// Mitsubishi GX Works2 project: plcV3   PLC: FX3G

TYPE ST_INTENS : STRUCT
  RECIRC : INT;
  ASPER : INT;
END_STRUCT END_TYPE

// global labels: GVL
VAR_GLOBAL
  g_iIntensity AT D500 : INT;  (* Интенсивность: 0=Слабо, 1=Нормально, 2=Интенсивно (настройка HMI) *)
  g_iToutAsper AT D501 : INT;  (* Мин. t улицы для аспирации, °C×10 (по умолч. 30 = 3.0°C) *)
  g_iToutHeat AT D502 : INT;  (* Мин. t улицы для подогрева, °C×10 (по умолч. 50 = 5.0°C) *)
  g_iPreheatTime AT D504 : INT;  (* Время предподогрева заслонок, мин (по умолч. 3) *)
  g_iManualAspMin AT D506 : INT;  (* Время ручной аспирации, мин (ввод оператора, по умолч. 5) *)
  g_iPreheatLeft AT D507 : INT;  (* Текущее время подогрева, мин (обратный отсчёт для HMI) *)
  g_iAutoResetDelay AT D508 : INT;  (* Задержка автосброса, мин (по умолч. 60) *)
  g_iTprodMax AT D509 : INT;  (* Макс. температура продукта, °C×10 (задаётся оператором) *)
  g_iHmin AT D510 : INT;  (* Мин. влажность, %×10 (задаётся оператором) *)
  g_iCorrTout AT D511 : INT;  (* Коррекция t улицы (Pt100), °C×10 (настройка HMI) *)
  g_iCorrTprod1 AT D512 : INT;  (* Коррекция щупа 1 (Pt100), °C×10 (настройка HMI) *)
  g_iCorrTprod2 AT D513 : INT;  (* Коррекция щупа 2 (Pt100), °C×10 (настройка HMI) *)
  g_iCorrTprod3 AT D514 : INT;  (* Коррекция щупа 3 (Pt100), °C×10 (настройка HMI) *)
  g_iCorrTprod4 AT D515 : INT;  (* Коррекция щупа 4 (Pt100), °C×10 (настройка HMI) *)
  g_iMbAddr AT D516 : INT;  (* Modbus slave: адрес ПЛК (1..247, по умолч. 1) *)
  g_iValveTime AT D517 : INT;  (* Время хода клапана, с (по умолч. 120) *)
  g_iProgress AT D518 : INT;  (* Время исполнения в % 0-100 *)
  g_iLeftTime AT D519 : INT;  (* Сколько минут осталось обратный отсчет *)
  g_iFun1State AT D520 : INT;  (* Состояние вентилятора 1 *)
  g_iFun2State AT D521 : INT;  (* Состояние вентилятора 2 *)
  g_iFun3State AT D522 : INT;  (* Состояние вентилятора 3 *)
  g_iFun4State AT D523 : INT;  (* Состояние вентилятора 4 *)
  g_iFun5State AT D524 : INT;  (* Состояние вентилятора 5 *)
  g_iFun6State AT D525 : INT;  (* Состояние вентилятора 6 *)
  g_iFun7State AT D526 : INT;  (* Состояние вентилятора 7 *)
  g_iFun8State AT D527 : INT;  (* Состояние вентилятора 8 *)
  g_iFun9State AT D528 : INT;  (* Состояние вентилятора 9 *)
  g_iFun10State AT D529 : INT;  (* Состояние вентилятора 10 *)
  g_iModeDisp AT D530 : INT;  (* Детальный режим для HMI: 0=Выкл, 1=Авто, 2=Продувка, 3=Аспирацияб, 4=Прогрев клапанов, 5-ручная аспирация *)
  g_iRecircLeft AT D531 : INT;  (* Отсчёт рециркуляции, мин *)
  g_iAspLeft AT D532 : INT;  (* Обратный отсчёт аспирации *)
  g_iAlarmCount AT D533 : INT;  (* Количество активных тревог *)
  g_iStep AT D534 : INT;  (* Состояние автомата (0/2/50/100/200/210/300, отладка) *)
  g_iModeCoarse AT D535 : INT;  (* Грубый режим по переключателю: 0=Выкл, 1=Авто, 2=Продувка *)
  g_iCurWait AT D536 : INT;  (* Текущее время ожидания в авто режиме в выбраной интенсивности *)
  g_iCurAsper AT D537 : INT;  (* Текущее время аспирации в авто режиме в выбраной интенсивности *)
  g_iAlarmPack1 AT D550 : INT;  (* Упакованные тревоги 0-15 (AM_PACK) *)
  g_iAlarmPack2 AT D551 : INT;  (* Упакованные тревоги 16-27 (AM_PACK) *)
  g_iAlarmPack3 AT D552 : INT;  (* Упакованные тревоги 32-33 (AM_PACK) *)
  g_xCmdFanH1 AT M500 : BOOL;  (* Команда напорный вентилятор 1 *)
  g_xCmdFanH2 AT M501 : BOOL;  (* Команда напорный вентилятор 2 *)
  g_xCmdFanH3 AT M502 : BOOL;  (* Команда напорный вентилятор 3 *)
  g_xCmdFanH4 AT M503 : BOOL;  (* Команда напорный вентилятор 4 *)
  g_xCmdFanH5 AT M504 : BOOL;  (* Команда напорный вентилятор 5 *)
  g_xCmdFanH6 AT M505 : BOOL;  (* Команда напорный вентилятор 6 *)
  g_xCmdFanR1 AT M506 : BOOL;  (* Команда разгонный вентилятор 1 *)
  g_xCmdFanR2 AT M507 : BOOL;  (* Команда разгонный вентилятор 2 *)
  g_xCmdFanR3 AT M508 : BOOL;  (* Команда разгонный вентилятор 3 *)
  g_xCmdFanR4 AT M509 : BOOL;  (* Команда разгонный вентилятор 4 *)
  g_xCmdValveIn1 AT M510 : BOOL;  (* Команда открыть клапан приток 1 *)
  g_xCmdValveIn2 AT M511 : BOOL;  (* Команда открыть клапан приток 2 *)
  g_xCmdValveOut1 AT M512 : BOOL;  (* Команда открыть клапан сброс 1 *)
  g_xCmdValveOut2 AT M513 : BOOL;  (* Команда открыть клапан сброс 2 *)
  g_xCmdValveRec1 AT M514 : BOOL;  (* Команда открыть клапан рециркуляция 1 *)
  g_xCmdValveRec2 AT M515 : BOOL;  (* Команда открыть клапан рециркуляция 2 *)
  g_xCmdHeat AT M516 : BOOL;  (* Подогрев клапана приток *)
  g_xCoolerWorks AT M517 : BOOL;  (* Холод работает *)
  g_xIsAuto AT M518 : BOOL;  (* Автоматический режим *)
  g_xAspirNow AT M519 : BOOL;  (* Сейчас идет асперация *)
  g_xCmdCoolerStop AT M520 : BOOL;  (* Команда «Остановить холод» (Y00) *)
  g_xManualAspActive AT M521 : BOOL;  (* Ручная аспирация выполняется *)
  g_xManualAspCmd AT M522 : BOOL;  (* Кнопка HMI: ручная аспирация (фронт) *)
  g_xAlarmResetHmi AT M523 : BOOL;  (* Кнопка HMI: сброс тревог (фронт) *)
  g_xModeManual AT M524 : BOOL;  (* Ручной режим если ни какой режим не выбран на входах *)
  g_xAutoReset AT M525 : BOOL;  (* Автосброс тревог: TRUE=вкл, FALSE=выкл (по умолч. выкл) *)
  g_xMbApply AT M526 : BOOL;  (* Кнопка HMI: применить настройки Modbus (фронт) *)
  g_xValveIn AT M527 : BOOL;  (* Кнопка HMI: применить настройки Modbus (фронт) *)
  g_xValveOut AT M528 : BOOL;  (* Кнопка HMI: применить настройки Modbus (фронт) *)
  g_xValveRecycle AT M529 : BOOL;  (* Кнопка HMI: применить настройки Modbus (фронт) *)
  g_xRecycleFlow AT M530 : BOOL;  (* Поток идет рециркуляция *)
  g_xAnyAlarm AT M550 : BOOL;  (* Есть активная тревога (AM_HAS_ALARMS) *)
  g_xAnyBlock AT M551 : BOOL;  (* Есть блокирующая тревога (AM_IS_BLOCK) *)
END_VAR
VAR_GLOBAL CONSTANT
  c_AM_ALARMS_NUM : INT := 33;  (* Верхняя граница массива AM_ALARMS (34 тревоги, ID 0..33) *)
  c_AM_EVENTS_NUM : INT;  (* Верхняя граница массива AM_EVENTS (события не используются) *)
END_VAR
VAR_GLOBAL
  astIntens : ARRAY [0..2] OF ST_INTENS;  (* Уровени интенсивности. Назначить D540 как главный *)
  AM_ALARMS : ARRAY [0..33] OF ST_AM_ALARM;  (* Хранилище тревог AlarmManager (объявляет приложение, V206+) *)
  AM_EVENTS : ARRAY [0..0] OF ST_AM_EVENT;  (* Хранилище событий AlarmManager (объявляет приложение, V206+) *)
  g_iTCorrection AT D538 : INT;  (* Корекция температуры *)
END_VAR

// global labels: IO
VAR_GLOBAL
  DI_ModeAuto AT X000 : BOOL;  (* Переключатель режима — «Авто» / ШУК-D1 *)
  DI_ModePurge AT X001 : BOOL;  (* Переключатель режима — «Продувка» / ШУК-D1 *)
  DI_PhaseFault AT X002 : BOOL;  (* Реле контроля фаз — ошибка фазировки / ШУК-D1 *)
  DI_CoolerRun AT X003 : BOOL;  (* Охладитель в работе (идёт охлаждение) / ШУК-D1 *)
  DI_VlvIn1Close AT X004 : BOOL;  (* Концевик клапана приток №1 — закрыт (НО) / ШУК-D1 *)
  DI_VlvIn2Close AT X005 : BOOL;  (* Концевик клапана приток №2 — закрыт (НО) / ШУК-D1 *)
  DI_FanHFb1 AT X006 : BOOL;  (* Обратная связь напорного вентилятора №1 (пускатель/тепловое реле) / ШУК-D1 *)
  DI_FanHFb2 AT X007 : BOOL;  (* Обратная связь напорного вентилятора №2 (пускатель/тепловое реле) / ШУК-D1 *)
  DI_FanHFb3 AT X010 : BOOL;  (* Обратная связь напорного вентилятора №3 (пускатель/тепловое реле) / ШУК-D1 *)
  DI_FanHFb4 AT X011 : BOOL;  (* Обратная связь напорного вентилятора №4 (пускатель/тепловое реле) / ШУК-D1 *)
  DI_FanHFb5 AT X012 : BOOL;  (* Обратная связь напорного вентилятора №5 (пускатель/тепловое реле) / ШУК-D1 *)
  DI_FanHFb6 AT X013 : BOOL;  (* Обратная связь напорного вентилятора №6 (пускатель/тепловое реле) / ШУК-D1 *)
  DI_VlvOut1Close AT X020 : BOOL;  (* Концевик клапана сброс №1 — закрыт (НО) / ШУК-D2 *)
  DI_VlvOut2Close AT X021 : BOOL;  (* Концевик клапана сброс №2 — закрыт (НО) / ШУК-D2 *)
  DI_VlvRec1Close AT X022 : BOOL;  (* Концевик клапана рециркуляция №1 — закрыт (НО) / ШУК-D2 *)
  DI_VlvRec2Close AT X023 : BOOL;  (* Концевик клапана рециркуляция №2 — закрыт (НО) / ШУК-D2 *)
  DI_VlvIn1Open AT X024 : BOOL;  (* Концевик клапана приток №1 — открыт / ШУК-D2 *)
  DI_VlvIn2Open AT X025 : BOOL;  (* Концевик клапана приток №2 — открыт / ШУК-D2 *)
  DI_VlvOut1Open AT X026 : BOOL;  (* Концевик клапана сброс №1 — открыт / ШУК-D2 *)
  DI_VlvOut2Open AT X027 : BOOL;  (* Концевик клапана сброс №2 — открыт / ШУК-D2 *)
  DI_VlvRec1Open AT X030 : BOOL;  (* Концевик клапана рециркуляция №1 — открыт / ШУК-D2 *)
  DI_VlvRec2Open AT X031 : BOOL;  (* Концевик клапана рециркуляция №2 — открыт / ШУК-D2 *)
  DI_Flow1 AT X032 : BOOL;  (* Реле давления №1 — поток есть / ШУК-D2; РД-ДД200, контакт НЗ *)
  DI_Flow2 AT X033 : BOOL;  (* Реле давления №2 — поток есть / ШУК-D2; РД-ДД200, контакт НЗ *)
  DI_Flow3 AT X034 : BOOL;  (* Реле давления №3 — поток есть / ШУК-D2; РД-ДД200, контакт НЗ *)
  DI_Flow4 AT X035 : BOOL;  (* Реле давления №4 — поток есть / ШУК-D2; РД-ДД200, контакт НЗ *)
  DI_Flow5 AT X036 : BOOL;  (* Реле давления №5 — поток есть / ШУК-D2; РД-ДД200, контакт НЗ *)
  DI_Flow6 AT X037 : BOOL;  (* Реле давления №6 — поток есть / ШУК-D2; РД-ДД200, контакт НЗ *)
  DO_CoolerStop AT Y000 : BOOL;  (* Остановить холод (1 = запрет охлаждения, 0 = разрешение) / ШУК-D1 *)
  DO_FanR1 AT Y002 : BOOL;  (* Разгонный вентилятор №1 (220 В, без обратной связи) / ШУК-D1 *)
  DO_FanR2 AT Y003 : BOOL;  (* Разгонный вентилятор №2 (220 В, без обратной связи) / ШУК-D1 *)
  DO_FanR3 AT Y004 : BOOL;  (* Разгонный вентилятор №3 (220 В, без обратной связи) / ШУК-D1 *)
  DO_FanR4 AT Y005 : BOOL;  (* Разгонный вентилятор №4 (220 В, без обратной связи) / ШУК-D1 *)
  DO_FanH1 AT Y006 : BOOL;  (* Напорный вентилятор №1 (2.2 кВт, 380 В) / ШУК-D1 *)
  DO_FanH2 AT Y007 : BOOL;  (* Напорный вентилятор №2 (2.2 кВт, 380 В) / ШУК-D1 *)
  DO_FanH3 AT Y010 : BOOL;  (* Напорный вентилятор №3 (2.2 кВт, 380 В) / ШУК-D1 *)
  DO_FanH4 AT Y011 : BOOL;  (* Напорный вентилятор №4 (2.2 кВт, 380 В) / ШУК-D1 *)
  DO_FanH5 AT Y012 : BOOL;  (* Напорный вентилятор №5 (2.2 кВт, 380 В) / ШУК-D1 *)
  DO_FanH6 AT Y013 : BOOL;  (* Напорный вентилятор №6 (2.2 кВт, 380 В) / ШУК-D1 *)
  DO_HeatVlv AT Y020 : BOOL;  (* Подогрев клапана (ТЭН 4x300 Вт) / ШУК-D3 *)
  DO_VlvIn1Open AT Y024 : BOOL;  (* Открыть клапан приток №1 (Belimo LF230, пружина закрывает) / ШУК-D3 *)
  DO_VlvIn2Open AT Y025 : BOOL;  (* Открыть клапан приток №2 (Belimo LF230, пружина закрывает) / ШУК-D3 *)
  DO_VlvOut1Open AT Y026 : BOOL;  (* Открыть клапан сброс №1 (Belimo LF230, пружина закрывает) / ШУК-D3 *)
  DO_VlvOut2Open AT Y027 : BOOL;  (* Открыть клапан сброс №2 (Belimo LF230, пружина закрывает) / ШУК-D3 *)
  DO_VlvRec1Open AT Y030 : BOOL;  (* Открыть клапан рециркуляция №1 (Belimo LF230, пружина закрывает) / ШУК-D3 *)
  DO_VlvRec2Open AT Y031 : BOOL;  (* Открыть клапан рециркуляция №2 (Belimo LF230, пружина закрывает) / ШУК-D3 *)
  DO_LampGreen AT Y032 : BOOL;  (* Световая колонна — зелёный / ШУК-D3 *)
  DO_LampRed AT Y033 : BOOL;  (* Световая колонна — красный / ШУК-D3 *)
  AI_fTOutside AT D0 : REAL;  (* t улицы (0-10 В), °C (REAL, натур. — FLT10 делит на 10) / ШУК-D1; °C×10 *)
  AI_fTChamber AT D2 : REAL;  (* t в камере (ПВТ110 4-20 мА), °C (REAL, натур. — FLT10 делит на 10) / ШУК-D1; °C×10 *)
  AI_fTProd1 AT D4 : REAL;  (* t продукта щуп 1 (Pt100, L02-RTD), °C (REAL, натур. — FLT10 делит на 10) / ШУК-D4; °C×10 *)
  AI_fTProd2 AT D6 : REAL;  (* t продукта щуп 2 (Pt100, L02-RTD), °C (REAL, натур. — FLT10 делит на 10) / ШУК-D4; °C×10 *)
  AI_fTProd3 AT D8 : REAL;  (* t продукта щуп 3 (Pt100, L02-RTD), °C (REAL, натур. — FLT10 делит на 10) / ШУК-D4; °C×10 *)
  AI_fTProd4 AT D10 : REAL;  (* t продукта щуп 4 (Pt100, L02-RTD), °C (REAL, натур. — FLT10 делит на 10) / ШУК-D4; °C×10 *)
  AI_fTProdAvg AT D12 : REAL;  (* Средняя t продукта (4 щупа), °C (REAL, натур.) / ШУК-D4; °C×10 *)
  AI_fHChamber AT D14 : REAL;  (* Влажность в камере (ПВТ110 4-20 мА), % (REAL, натур. — FLT10 делит на 10) / ШУК-D1; %×10 *)
  AI_iRawTChamber AT D8032 : INT;  (* Сырое значение t в камере (для обрыва 4-20 мА, ≥ 32720) / ШУК-D1 *)
  AI_iRawHChamber AT D8033 : INT;  (* Сырое значение влажности (для обрыва 4-20 мА, ≥ 32720) / ШУК-D1 *)
END_VAR

// task Task_01 (event TRUE, interval 0, priority 31): MAIN
// task TCO (event I750, interval 0, priority 2): PRG_TCO_TICKER_50
// task INIT (event M8002, interval 0, priority 1): INIT
// task ROUTINE (event FALSE, interval T#100ms, priority 30): ROUTINE
// user libraries (not included): AlarmManager, Modbus, TimeControl, Utils

PROGRAM MAIN
VAR
  iState : INT;  (* State of the automaton (0/2/50/100/200/210/300) *)
  iPrevState : INT;  (* Previous state (for edge detection) *)
  xEntry : BOOL;  (* Entry edge flag (single-scan on state change) *)
  iAspTarget : INT;  (* Aspiration duration target, min (regular or manual) *)
  fbTON1 : TON;  (* On-delay: FanH1 (2 s) *)
  fbTON2 : TON;  (* On-delay: FanH2 (4 s) *)
  fbTON3 : TON;  (* On-delay: FanH3 (6 s) *)
  fbTON4 : TON;  (* On-delay: FanH4 (8 s) *)
  fbTON5 : TON;  (* On-delay: FanH5 (10 s) *)
  fbTON6 : TON;  (* On-delay: FanH6 (12 s) *)
  fbTON7 : TON;  (* On-delay: FanR1 (14 s) *)
  fbTON8 : TON;  (* On-delay: FanR2 (16 s) *)
  fbTON9 : TON;  (* On-delay: FanR3 (18 s) *)
  fbTON10 : TON;  (* On-delay: FanR4 (20 s) *)
  STATE_RESET : INT;  (* State constant: 0 *)
  STATE_IDLE : INT;  (* State constant: 2 *)
  STATE_PURGE : INT;  (* State constant: 50 *)
  STATE_RECIRC : INT;  (* State constant: 100 *)
  STATE_PREPARE : INT;  (* State constant: 200 *)
  STATE_PREHEAT : INT;  (* State constant: 210 *)
  STATE_ASPER : INT;  (* State constant: 300 *)
  fbTOF1 : TOF;  (* Off-delay: FanH1 (onпорный 1) *)
  fbTOF2 : TOF;  (* Off-delay: FanH2 (onпорный 2) *)
  fbTOF3 : TOF;  (* Off-delay: FanH3 (onпорный 3) *)
  fbTOF4 : TOF;  (* Off-delay: FanH4 (onпорный 4) *)
  fbTOF5 : TOF;  (* Off-delay: FanH5 (onпорный 5) *)
  fbTOF6 : TOF;  (* Off-delay: FanH6 (onпорный 6) *)
  fbTOF7 : TOF;  (* Off-delay: FanR1 (разгонный 1) *)
  fbTOF8 : TOF;  (* Off-delay: FanR2 (разгонный 2) *)
  fbTOF9 : TOF;  (* Off-delay: FanR3 (разгонный 3) *)
  fbTOF10 : TOF;  (* Off-delay: FanR4 (разгонный 4) *)
  fbTOF11 : TOF;  (* Off-delay: VlvIn1 (клапан приток 1) *)
  fbTOF12 : TOF;  (* Off-delay: VlvIn2 (клапан приток 2) *)
  fbTOF13 : TOF;  (* Off-delay: VlvOut1 (клапан сброс 1) *)
  fbTOF14 : TOF;  (* Off-delay: VlvOut2 (клапан сброс 2) *)
  fbTOF15 : TOF;  (* Off-delay: VlvRec1 (клапан рециркуляция 1) *)
  fbTOF16 : TOF;  (* Off-delay: VlvRec2 (клапан рециркуляция 2) *)
END_VAR
(*
  MAIN — главная программа (Program): БИЗНЕС-ЛОГИКА
  Проект: автоматизация камеры овощехранилища (ШУК.260726), ПЛК COOLMAY-L02
  Среда: GX Works 2, IEC 61131-3 Structured Text

  ФБ FB_PROCESS и FB_ACTUATORS УДАЛЕНЫ — их код вставлен в эту программу
  напрямую и объединён:
    1) конечный автомат режима «Авто» (рециркуляция / аспирация /
       ручная аспирация) + выбор грубого режима по переключателю;
    2) приводы: клапаны, вентиляторы, подогрев, блокировка охладителя Y00.

  Рутины (аналоговые входы, тревоги, световая колонна) вынесены в
  отдельную программу PRG_ROUTINE. Порядок выполнения программ в задаче:
  PRG_ROUTINE → PRG_MAIN (данные/тревоги до бизнес-логики).

  Программа INIT запускается отдельно, один раз при старте (см. PRG_INIT.st).
  HMI TK8100 читает входы/выходы и D/M-регистры напрямую — отдельного
  блока статусов HMI не требуется.

  Локальные переменные — в PRG_MAIN.csv.
 *)

(* Разрешение прерываний (EI) — первая строка каждой программы *)
EI(TRUE);

(* ════════════════════════════════════════════════════════════════
   ЧАСТЬ 1. КОНЕЧНЫЙ АВТОМАТ (код бывшего FB_PROCESS)
   ════════════════════════════════════════════════════════════════
   Состояния (g_iStep, D534 — для отладки/HMI):
      0 — СБРОС (однократный сброс выходов, безусловный переход в 2)
      2 — ОЖИДАНИЕ (Выключено; ожидание команды режима)
     50 — ПРОДУВКА (рециркуляция открыта, вентиляторы — вручную)
    100 — РЕЦИРКУЛЯЦИЯ (основное состояние)
    200 — ПОДГОТОВКА К АСПИРАЦИИ (проверка t улицы, решение: подогрев или сразу аспирация)
    210 — ПОДОГРЕВ ЗАСЛОНОК (греем ТЭН клапанов приток/сброс, потом открываем клапаны, включаем все вент., запускаем аспирацию)
    300 — АСПИРАЦИЯ (все 10 вент. уже включены в 210, только обратный отсчёт)

  Структура (по решению ревью): шаг 0 — только сброс, безусловно → 2;
  шаг 2 (ОЖИДАНИЕ) ждёт команду режима: Продувка → 50, Авто → 100,
  ручная аспирация → 200; при «Выключено» остаёмся в 2.
  Выход из «Авто» (100–300) при сигнале «не Авто» → шаг 0 → 2.

  Логика по плану §6.4:
  - рециркуляция: длительность по интенсивности (1200/600/300 мин),
    клапаны рециркуляции открыты, Y00 = 0; вентиляторы следуют за X03
    (охладитель) — реализовано ниже, в части «Приводы»;
  - перед аспирацией проверка t улицы: при t ≤ g_iToutAsper — пропуск
    цикла (слишком холодно); при t ≤ g_iToutHeat — подогрев заслонок;
  - аспирация 5 мин (300 с, регулярная) или g_iManualAspMin (ручная);
  - Y00 = 1 только во время аспирации (запрет охлаждения).

  Ручная аспирация (HMI: g_xManualAspCmd + g_iManualAspMin):
  - приоритет над регулярной; работает из любого режима;
  - по завершении возврат: в Авто — в рециркуляцию, иначе — в ОЖИДАНИЕ (2).

  Блокирующая тревога (g_xAnyBlock — реле фаз) НЕ останавливает автомат:
  блокируются только напорные вентиляторы (380 В). Разгонные (220 В)
  реле контроля фаз не затрагивает (ТЗ §7.6, v1.2).
 *)

(* Грубый выбор режима по переключателю
0 - Off
1 - Рециркуляция
2 - Продувка
 *)
g_iModeCoarse := SEL(DI_ModePurge, SEL(DI_ModeAuto, 0, 1), 2);

(* для HMI: 0=Выкл, 1=Рециркуляция, 2=Продувка, 3=Аспирация, 4=Прогрев клапанов *)
g_iModeDisp := g_iModeCoarse;
MOV(iState >= 200, 3, g_iModeDisp); (* Аспирация: 200 подготовка, 300 аспирация *)
MOV(iState = 210, 4, g_iModeDisp); (* Прогрев клапанов *)
MOV(iState >= 200 AND g_xManualAspActive, 5, g_iModeDisp); (* Асперация в ручном режиме *)

(* Если выключили во время аспирации *)
MOV(g_iModeCoarse = 0 AND iState >= 200, STATE_RESET, iState);

(* ── Фронт входа в состояние (однократные действия) ──────────── *)
xEntry := MEP(iState <> iPrevState);
iPrevState := iState;

(* Ручная аспирация из Выключено (возврат в этот же режим) *)
IF MEP(g_xManualAspCmd) THEN
    IF g_iModeDisp = 1 THEN
        g_xManualAspActive := TRUE;
        iState := STATE_PREPARE; (* подготовка к аспирации *)
    ELSE
        g_xManualAspCmd := FALSE; (* игнор команды, если уже в аспирации *)
    END_IF;
END_IF;

STATE_RESET := 0;
STATE_IDLE := 2;
STATE_PURGE := 50;
STATE_RECIRC := 100;
STATE_PREPARE := 200;
STATE_PREHEAT := 210;
STATE_ASPER := 300;

(* 0=низкая, 1=средняя, 2=высокая *)
g_iIntensity := LIMITATION(0, g_iIntensity, 2);

CASE iState OF
0: (* СБРОС: все выходы в безопасное состояние, безусловно → 2 *)
    (* Вентиляторы выключены, клапаны закрыты, подогрев выключен,
       холод не блокируется *)
    g_xCmdFanH1 := FALSE; g_xCmdFanH2 := FALSE;
    g_xCmdFanH3 := FALSE; g_xCmdFanH4 := FALSE;
    g_xCmdFanH5 := FALSE; g_xCmdFanH6 := FALSE;
    g_xCmdFanR1 := FALSE; g_xCmdFanR2 := FALSE;
    g_xCmdFanR3 := FALSE; g_xCmdFanR4 := FALSE;
    g_xCmdValveIn1 := FALSE; g_xCmdValveIn2 := FALSE;
    g_xCmdValveOut1 := FALSE; g_xCmdValveOut2 := FALSE;
    g_xCmdValveRec1 := FALSE; g_xCmdValveRec2 := FALSE;
    g_xCmdHeat := FALSE;
    g_xCmdCoolerStop := FALSE;
    g_xManualAspActive := FALSE;
    g_xValveIn := FALSE; g_xValveOut := FALSE; g_xValveRecycle := FALSE;

    g_iPreheatLeft := 0; g_iAspLeft := 0; g_iRecircLeft := 0;
    g_xManualAspCmd := FALSE; (* сброс фронта ручной аспирации *)

    iState := STATE_IDLE; (* безусловный переход в ОЖИДАНИЕ *)

2: (* ОЖИДАНИЕ Выключено: ждём команду режима *)
    (* Команды режима: Продувка → 50, Авто → 100 *)
    IF g_iModeCoarse = 1 THEN
        iState := STATE_RECIRC;
    ELSIF g_iModeCoarse = 2 THEN
        iState := STATE_PURGE;
    END_IF;

    IF iState <> STATE_IDLE THEN
        g_xCmdFanH1 := FALSE; g_xCmdFanH2 := FALSE;
        g_xCmdFanH3 := FALSE; g_xCmdFanH4 := FALSE;
        g_xCmdFanH5 := FALSE; g_xCmdFanH6 := FALSE;
        g_xCmdFanR1 := FALSE; g_xCmdFanR2 := FALSE;
        g_xCmdFanR3 := FALSE; g_xCmdFanR4 := FALSE;
        g_xCmdValveIn1 := FALSE; g_xCmdValveIn2 := FALSE;
        g_xCmdValveOut1 := FALSE; g_xCmdValveOut2 := FALSE;
        g_xCmdValveRec1 := FALSE; g_xCmdValveRec2 := FALSE;
        g_xCmdHeat := FALSE;
        g_xCmdCoolerStop := FALSE;
        g_xManualAspActive := FALSE;
        g_xValveIn := FALSE; g_xValveOut := FALSE; g_xValveRecycle := FALSE;
    END_IF;

50: (* ПРОДУВКА: рециркуляция открыта, вентиляторы — вручную *)
    (* Команды режима: Выключено → через сброс в ОЖИДАНИЕ, Авто → 100 *)
    g_xCmdFanH1 := TRUE; g_xCmdFanH2 := TRUE;
    g_xCmdFanH3 := TRUE; g_xCmdFanH4 := TRUE;
    g_xCmdFanH5 := TRUE; g_xCmdFanH6 := TRUE;
    g_xCmdFanR1 := TRUE; g_xCmdFanR2 := TRUE;
    g_xCmdFanR3 := TRUE; g_xCmdFanR4 := TRUE;

    (* Клапаны: рециркуляция открыта, приток/сброс закрыты *)
    g_xCmdValveRec1 := TRUE; g_xCmdValveRec2 := TRUE;

    IF g_iModeCoarse <> 2 THEN
        iState := STATE_RESET;
    END_IF;

100: (* РЕЦИРКУЛЯЦИЯ *)
    g_xCmdFanH1 := DI_CoolerRun; g_xCmdFanH2 := DI_CoolerRun;
    g_xCmdFanH3 := DI_CoolerRun; g_xCmdFanH4 := DI_CoolerRun;
    g_xCmdFanH5 := DI_CoolerRun; g_xCmdFanH6 := DI_CoolerRun;
    g_xCmdFanR1 := DI_CoolerRun; g_xCmdFanR2 := DI_CoolerRun;
    g_xCmdFanR3 := DI_CoolerRun; g_xCmdFanR4 := DI_CoolerRun;

    (* Клапаны: рециркуляция открыта, приток/сброс закрыты *)
    g_xCmdValveRec1 := TRUE; g_xCmdValveRec2 := TRUE;

    IF g_iModeCoarse <> 1 THEN
        iState := STATE_RESET;
    END_IF;

    (* Тик 1 мин (M8014) — обратный отсчёт рециркуляции *)
    INCP(M8014, g_iRecircLeft);
    IF g_iRecircLeft >= astIntens[g_iIntensity].RECIRC THEN
        g_iRecircLeft := 0; (* сброс счётчика рециркуляции *)
        iState := STATE_PREPARE;
    END_IF;

200: (* ПОДГОТОВКА К АСПИРАЦИИ *)
    IF AI_fTOutside <= F_FLT10(g_iToutHeat) THEN
        g_xCmdHeat := TRUE;
        iState := STATE_PREHEAT; (* Подогрев *)
    ELSE
        iState := STATE_ASPER; (* Аспирация *)
    END_IF;

    IF g_xManualAspActive THEN
        iAspTarget := g_iManualAspMin; (* ручная аспирация: мин. время *)
    ELSE
        iAspTarget := astIntens[g_iIntensity].ASPER; (* регулярная аспирация: 5 мин *)
    END_IF;

    (* Если температура outside не превышает порог аспирации не будет иначе заморозим продукт *)
    IF AI_fTOutside <= F_FLT10(g_iToutAsper) THEN
        g_xCmdHeat := FALSE;
        iState := STATE_RESET;
    END_IF;

210: (* ПОДОГРЕВ ЗАСЛОНОК *)
    INCP(M8014, g_iPreheatLeft);
    IF g_iPreheatLeft >= g_iPreheatTime THEN
        g_iPreheatLeft := 0; (* сброс счётчика подогрева *)

        (* Подогрев выключен *)
        g_xCmdHeat := FALSE;

        iState := STATE_ASPER; (* Аспирация *)
    END_IF;

300: (* АСПИРАЦИЯ: все 10 вент., приток/сброс открыты, рециркуляция закрыта *)
(* Холод остановлен *)
    g_xCmdCoolerStop := TRUE;

    (* Вентиляторы: все 10 включены *)
    g_xCmdFanH1 := TRUE; g_xCmdFanH2 := TRUE;
    g_xCmdFanH3 := TRUE; g_xCmdFanH4 := TRUE;
    g_xCmdFanH5 := TRUE; g_xCmdFanH6 := TRUE;
    g_xCmdFanR1 := TRUE; g_xCmdFanR2 := TRUE;
    g_xCmdFanR3 := TRUE; g_xCmdFanR4 := TRUE;

    (* Клапаны: приток/сброс открыть, рециркуляцию закрыть *)
    g_xCmdValveIn1 := TRUE; g_xCmdValveIn2 := TRUE;
    g_xCmdValveOut1 := TRUE; g_xCmdValveOut2 := TRUE;
    g_xCmdValveRec1 := FALSE; g_xCmdValveRec2 := FALSE;

    (* Выход из Авто → сброс *)
    IF g_iModeCoarse <> 1 THEN
        iState := STATE_RESET;
    END_IF;

    (* Обратный отсчёт аспирации *)
    INCP(M8014, g_iAspLeft);
    IF g_iAspLeft >= iAspTarget THEN
        g_iAspLeft := 0; (* сброс счётчика *)
        iState := STATE_RESET; (* завершение аспирации → сброс *)
    END_IF;

ELSE
    (* Неизвестное состояние — сброс в шаг 0 (СБРОС), страховка *)
    iState := 0;
END_CASE;

(* Номер состояния автомата — для отладки и HMI *)
g_iStep := iState;

(* ════════════════════════════════════════════════════════════════
   ЧАСТЬ 1.5. ПРОГРЕСС И ОСТАВШЕЕСЯ ВРЕМЯ (для HMI)
   g_iProgress — 0..100 % выполнения текущей фазы (рециркуляция/прогрев/аспирация);
   g_iLeftTime — сколько минут осталось до конца текущей фазы.

   Длительности фаз:
   - рециркуляция: astIntens[g_iIntensity].RECIRC (мин);
   - прогрев: g_iPreheatTime, мин (счётчик g_iPreheatLeft);
   - аспирация: astIntens[g_iIntensity].ASPER (мин, регулярная) либо
                   g_iManualAspMin (ручная) — уже в локальном iAspTarget.

   Счётчики g_iRecircLeft / g_iPreheatLeft / g_iAspLeft считают ВВЕРХ
   (INCP по тику M8014, 1 мин), поэтому «осталось» = длительность − счётчик,
   «прогресс» = счётчик ÷ длительность × 100 %. В прочих состояниях
   (Выкл, Продувка, подготовка) — 0 % и 0 мин.
   ════════════════════════════════════════════════════════════════ *)
CASE iState OF
    100: (* РЕЦИРКУЛЯЦИЯ *)
        IF astIntens[g_iIntensity].RECIRC > 0 THEN
            g_iProgress := REAL_TO_INT(INT_TO_REAL(g_iRecircLeft) * 100.0
                                       / INT_TO_REAL(astIntens[g_iIntensity].RECIRC));
            g_iLeftTime := astIntens[g_iIntensity].RECIRC - g_iRecircLeft;
        ELSE
            g_iProgress := 0;
            g_iLeftTime := 0;
        END_IF;
    210: (* ПРОГРЕВ КЛАПАНОВ *)
        IF g_iPreheatTime > 0 THEN
            g_iProgress := REAL_TO_INT(INT_TO_REAL(g_iPreheatLeft) * 100.0
                                       / INT_TO_REAL(g_iPreheatTime));
            g_iLeftTime := g_iPreheatTime - g_iPreheatLeft;
        ELSE
            g_iProgress := 0;
            g_iLeftTime := 0;
        END_IF;
    300: (* АСПИРАЦИЯ *)
        IF iAspTarget > 0 THEN
            g_iProgress := REAL_TO_INT(INT_TO_REAL(g_iAspLeft) * 100.0
                                       / INT_TO_REAL(iAspTarget));
            g_iLeftTime := iAspTarget - g_iAspLeft;
        ELSE
            g_iProgress := 0;
            g_iLeftTime := 0;
        END_IF;
    ELSE
        g_iProgress := 0;
        g_iLeftTime := 0;
END_CASE;

(* ════════════════════════════════════════════════════════════════
   ЧАСТЬ 2. ПРИВОДЫ (код бывшего FB_ACTUATORS)
   ════════════════════════════════════════════════════════════════
   - напорные вентиляторы Y06–Y13 (6 шт.);
   - разгонные вентиляторы Y02–Y05 (4 шт., 220 В);
   - клапаны Belimo Y24–Y31 (питание = открыть, пружина = закрыть);
   - подогрев заслонок Y20–Y23 (4 ТЭН);
   - блокировка охладителя Y00 (1 = запрет охлаждения, 0 = разрешение).

   Особенности:
   - в режиме «Рециркуляция» (g_iModeDisp = 1) все вентиляторы следуют
     за охладителем X03 (ТЗ §7.3.1);
   - блокирующая тревога «реле фаз» (g_xAnyBlock) снимает команды
     ТОЛЬКО напорных вентиляторов (380 В); разгонные (220 В, 1-фазн.)
     РКФ не блокирует (ТЗ §7.6, v1.2);
   - в «Продувке» вентиляторами управляет оператор вручную — команды
     автомата в этом режиме равны FALSE (см. выше, состояние ПРОДУВКА).
 *)

(* ── Вентиляторы: каскадный пуск с интервалом 2 с ─────────────── *)
(* У каждого вентилятора СВОЙ таймер задержки включения (TON),
   отсчитываемый от фронта его собственной команды: FanH1 — 2 с,
   FanH2 — 4 с, ... FanR4 — 20 с. Так каскад работает одинаково и в
   Авто (все команды приходят разом), и в ручном режиме (вентиляторы
   включают по одному — каждый ждёт свою ступень, а не включается
   мгновенно). Выключение — сразу у всех; TOF держит выход ещё 3 с.

   РУЧНОЙ РЕЖИМ (Выключено, g_xModeManual = TRUE, iState = 2 = STATE_IDLE):
   каскад TON гасится (AND NOT g_xModeManual), а выход вентилятора берётся
   напрямую из команды g_xCmdFan* (M500–M509) БЕЗ TOF — мгновенное
   включение и выключение (см. SEL ниже).
   Условие (iState = STATE_IDLE) в ручной ветке защищает от гонки:
   в скане перехода Продувка/Авто -> Выключено iState уже 0
   (STATE_RESET), а не 2, поэтому ещё не сброшенные команды автомата
   (g_xCmdFan* = TRUE) НЕ проходят в ручную ветку и не включают
   вентиляторы все разом. *)
g_xModeManual := NOT DI_ModeAuto AND NOT DI_ModePurge; (* для HMI: ручной режим вентиляторов *)

fbTON1(IN := g_xCmdFanH1 AND NOT g_xModeManual, PT := T#2s);
fbTON2(IN := g_xCmdFanH2 AND NOT g_xModeManual, PT := T#4s);
fbTON3(IN := g_xCmdFanH3 AND NOT g_xModeManual, PT := T#6s);
fbTON4(IN := g_xCmdFanH4 AND NOT g_xModeManual, PT := T#8s);
fbTON5(IN := g_xCmdFanH5 AND NOT g_xModeManual, PT := T#10s);
fbTON6(IN := g_xCmdFanH6 AND NOT g_xModeManual, PT := T#12s);
fbTON7(IN := g_xCmdFanR1 AND NOT g_xModeManual, PT := T#14s);
fbTON8(IN := g_xCmdFanR2 AND NOT g_xModeManual, PT := T#16s);
fbTON9(IN := g_xCmdFanR3 AND NOT g_xModeManual, PT := T#18s);
fbTON10(IN := g_xCmdFanR4 AND NOT g_xModeManual, PT := T#20s);


fbTOF1(IN := fbTON1.Q, PT := T#3s);
fbTOF2(IN := fbTON2.Q, PT := T#3s);
fbTOF3(IN := fbTON3.Q, PT := T#3s);
fbTOF4(IN := fbTON4.Q, PT := T#3s);
fbTOF5(IN := fbTON5.Q, PT := T#3s);
fbTOF6(IN := fbTON6.Q, PT := T#3s);
fbTOF7(IN := fbTON7.Q, PT := T#3s);
fbTOF8(IN := fbTON8.Q, PT := T#3s);
fbTOF9(IN := fbTON9.Q, PT := T#3s);
fbTOF10(IN := fbTON10.Q, PT := T#3s);

(* Выходы вентиляторов:
   - Авто/Продувка (g_xModeManual = FALSE): каскад TON + TOF 3 с;
   - Выключено, устойчивое (g_xModeManual = TRUE И iState = STATE_IDLE):
     ручная команда напрямую, БЕЗ TOF(мгновенное вкл/выкл);
   - переходный скан (g_xModeManual = TRUE, iState = 0): fbTOF*.Q —
     додержать каскадные, не включать новые (защита от гонки). *)
DO_FanH1 := SEL(g_xModeManual AND (iState = STATE_IDLE), fbTOF1.Q, g_xCmdFanH1);
DO_FanH2 := SEL(g_xModeManual AND (iState = STATE_IDLE), fbTOF2.Q, g_xCmdFanH2);
DO_FanH3 := SEL(g_xModeManual AND (iState = STATE_IDLE), fbTOF3.Q, g_xCmdFanH3);
DO_FanH4 := SEL(g_xModeManual AND (iState = STATE_IDLE), fbTOF4.Q, g_xCmdFanH4);
DO_FanH5 := SEL(g_xModeManual AND (iState = STATE_IDLE), fbTOF5.Q, g_xCmdFanH5);
DO_FanH6 := SEL(g_xModeManual AND (iState = STATE_IDLE), fbTOF6.Q, g_xCmdFanH6);
DO_FanR1 := SEL(g_xModeManual AND (iState = STATE_IDLE), fbTOF7.Q, g_xCmdFanR1);
DO_FanR2 := SEL(g_xModeManual AND (iState = STATE_IDLE), fbTOF8.Q, g_xCmdFanR2);
DO_FanR3 := SEL(g_xModeManual AND (iState = STATE_IDLE), fbTOF9.Q, g_xCmdFanR3);
DO_FanR4 := SEL(g_xModeManual AND (iState = STATE_IDLE), fbTOF10.Q, g_xCmdFanR4);

DO_FanH1 := DO_FanH1 AND NOT g_xAnyBlock AND g_iFun1State < 2;
DO_FanH2 := DO_FanH2 AND NOT g_xAnyBlock AND g_iFun2State < 2;
DO_FanH3 := DO_FanH3 AND NOT g_xAnyBlock AND g_iFun3State < 2;
DO_FanH4 := DO_FanH4 AND NOT g_xAnyBlock AND g_iFun4State < 2;
DO_FanH5 := DO_FanH5 AND NOT g_xAnyBlock AND g_iFun5State < 2;
DO_FanH6 := DO_FanH6 AND NOT g_xAnyBlock AND g_iFun6State < 2;

(* ── Клапаны (Belimo: питание = открыть, пружина = закрыть) ───── *)
fbTOF11(IN := g_xCmdValveIn1, PT := T#3s);
fbTOF12(IN := g_xCmdValveIn2, PT := T#3s);
fbTOF13(IN := g_xCmdValveOut1, PT := T#3s);
fbTOF14(IN := g_xCmdValveOut2, PT := T#3s);
fbTOF15(IN := g_xCmdValveRec1, PT := T#3s);
fbTOF16(IN := g_xCmdValveRec2, PT := T#3s);

DO_VlvIn1Open := SEL(g_xModeManual AND (iState = STATE_IDLE), fbTOF11.Q, g_xValveIn);
DO_VlvIn2Open := SEL(g_xModeManual AND (iState = STATE_IDLE), fbTOF12.Q, g_xValveIn);
DO_VlvOut1Open := SEL(g_xModeManual AND (iState = STATE_IDLE), fbTOF13.Q, g_xValveOut);
DO_VlvOut2Open := SEL(g_xModeManual AND (iState = STATE_IDLE), fbTOF14.Q, g_xValveOut);
DO_VlvRec1Open := SEL(g_xModeManual AND (iState = STATE_IDLE), fbTOF15.Q, g_xValveRecycle);
DO_VlvRec2Open := SEL(g_xModeManual AND (iState = STATE_IDLE), fbTOF16.Q, g_xValveRecycle);

(* ── Подогрев заслонок приток/сброс ──────────────────────────── *)
DO_HeatVlv := g_xCmdHeat;

(* ── Блокировка охладителя: 1 = запрет, 0 = разрешение ───────── *)
DO_CoolerStop := g_xCmdCoolerStop;
END_PROGRAM

PROGRAM INIT
VAR
  fbAMInit : FB_AM_INIT;  (* Конфигурация тревог AlarmManager V212 (34 вызова) *)
  PortSetting : DWORD;
END_VAR
(*
  INIT — отдельная программа однократной инициализации (Program)
  ЗАПУСКАЕТСЯ ОДИН РАЗ при старте ПЛК (первый скан / M8002 в настройках
  задачи). НЕ вызывается из MAIN и НЕ оборачивается в IF M8002.
  Если задача запускается циклически — вернуть обёртку IF M8002,
  иначе настройки и FB_AM_INIT будут выполняться каждый скан.

  Содержимое:
  - настройки по умолчанию — применяются ТОЛЬКО если текущее значение = 0
    (первый старт / после сброса регистров); изменения с HMI сохраняются
    между перезапусками ПЛК;
  - AlarmManager V212: конфигурация 34 тревог (FB_AM_INIT); хранилище AM_ALARMS объявлено в GVL (c_AM_ALARMS_NUM = 33);
  - Modbus slave (порт 2, RS-485) инициализируется в PRG_ROUTINE (не здесь).

  IP-адрес ПЛК с HMI больше не настраивается (регистры D520–D523 упразднены —
  теперь это состояния вентиляторов g_iFun1State..g_iFun4State).

  Локальные переменные — в PRG_INIT.csv (класс VAR, Program).
*)

(* Разрешение прерываний (EI) — первая строка каждой программы *)
EI(TRUE);

D8058 := 2#0000_0000_0000_1100;


(* ── Настройки по умолчанию (ТЗ §8.5) ───────────────────────
   Правило: уставка проставляется ТОЛЬКО если текущее значение = 0
   И сама уставка > 0. Это значит, что настройки, изменённые оператором
   с HMI, сохраняются между перезапусками ПЛК; заводские значения
   применяются лишь при первом старте (или после сброса D-регистров).
   Следствие: уставку нельзя сознательно задать равной 0 (например,
   ToutMin = 0.0 °C) — при перезапуске она вернётся к заводскому
   значению. Для уставок по умолчанию 0 (TprodMax, Hmin, коррекции)
   запись не выполняется вообще — они остаются как есть. *)

IF g_iIntensity = 0 THEN g_iIntensity := 2; END_IF;   (* 600 мин рециркуляции *)
IF g_iToutAsper = 0 THEN g_iToutAsper := 30; END_IF;  (* 3.0 °C — мин. t улицы для аспирации *)
IF g_iToutHeat = 0 THEN g_iToutHeat := 50; END_IF;   (* 5.0 °C — мин. t улицы для подогрева заслонок *)
IF g_iPreheatTime = 0 THEN g_iPreheatTime := 3; END_IF;   (* 3 мин — предподогрев *)
IF g_iManualAspMin = 0 THEN g_iManualAspMin := 5; END_IF; (* 5 мин — ручн. аспирация *)
(* g_xAutoReset: BOOL, заводское FALSE — не трогаем; выбор оператора
   (вкл/выкл) сохраняется между перезапусками. *)
IF g_iAutoResetDelay = 0 THEN g_iAutoResetDelay := 120; END_IF; (* 60 мин — автосброс *)
(* g_iTprodMax, g_iHmin: заводская уставка 0, задаётся оператором с HMI —
   не перезаписываем, иначе нельзя сохранить 0 (запрет тревог). *)
(* Коррекция датчиков Pt100 (HMI, °C×10): заводская уставка 0 —
   не перезаписываем (настройка оператора). *)

(* Настройки Modbus slave (порт 2): заводские значения применяются
   только если текущее значение = 0; изменения с HMI сохраняются. *)
IF g_iMbAddr = 0 THEN g_iMbAddr := 1; END_IF;        (* адрес 1 *)
IF g_iValveTime = 0 THEN g_iValveTime := 120; END_IF; (* 120 с — ход клапана *)

(* ── AlarmManager V212: конфигурация тревог (34 шт.) ────────
   Нумерация 0–33, задержки в единицах 50 мс (тик TCO_TICKER_50).
   См. план §5.
   ВАЖНО (V206+): хранилище AM_ALARMS/AM_EVENTS и константы ёмкости
   c_AM_ALARMS_NUM/c_AM_EVENTS_NUM объявляет ПРИЛОЖЕНИЕ (в GVL.csv),
   библиотека их больше не резервирует — строки «AM_ALARMS_NUM := 28» нет. *)

(* 0: реле контроля фаз — Error, мгновенно, блокирующая (стоп моторов) *)
fbAMInit(iNum := 0, iSeverity := c_AM_ERROR, iProcess := 1, iDelay := 0,
         xLock := TRUE, xLatch := FALSE, xBuzzer := FALSE);

(* 1–6: клапан не открылся — Warning, 60 с (iDelay g_iValveTime (сек) / 20 = х50 мс) *)
fbAMInit(iNum := 1, iSeverity := c_AM_WARNING, iProcess := 1, iDelay := g_iValveTime / 20,
         xLock := FALSE, xLatch := FALSE, xBuzzer := FALSE);
fbAMInit(iNum := 2, iSeverity := c_AM_WARNING, iProcess := 1, iDelay := g_iValveTime / 20,
         xLock := FALSE, xLatch := FALSE, xBuzzer := FALSE);
fbAMInit(iNum := 3, iSeverity := c_AM_WARNING, iProcess := 1, iDelay := g_iValveTime / 20,
         xLock := FALSE, xLatch := FALSE, xBuzzer := FALSE);
fbAMInit(iNum := 4, iSeverity := c_AM_WARNING, iProcess := 1, iDelay := g_iValveTime / 20,
         xLock := FALSE, xLatch := FALSE, xBuzzer := FALSE);
fbAMInit(iNum := 5, iSeverity := c_AM_WARNING, iProcess := 1, iDelay := g_iValveTime / 20,
         xLock := FALSE, xLatch := FALSE, xBuzzer := FALSE);
fbAMInit(iNum := 6, iSeverity := c_AM_WARNING, iProcess := 1, iDelay := g_iValveTime / 20,
         xLock := FALSE, xLatch := FALSE, xBuzzer := FALSE);

(* 7–12: нет потока воздуха, напорный вентилятор — Error, 30 с (iDelay 600 × 50 мс) *)
fbAMInit(iNum := 7, iSeverity := c_AM_ERROR, iProcess := 1, iDelay := 600,
         xLock := FALSE, xLatch := FALSE, xBuzzer := FALSE);
fbAMInit(iNum := 8, iSeverity := c_AM_ERROR, iProcess := 1, iDelay := 600,
         xLock := FALSE, xLatch := FALSE, xBuzzer := FALSE);
fbAMInit(iNum := 9, iSeverity := c_AM_ERROR, iProcess := 1, iDelay := 600,
         xLock := FALSE, xLatch := FALSE, xBuzzer := FALSE);
fbAMInit(iNum := 10, iSeverity := c_AM_ERROR, iProcess := 1, iDelay := 600,
         xLock := FALSE, xLatch := FALSE, xBuzzer := FALSE);
fbAMInit(iNum := 11, iSeverity := c_AM_ERROR, iProcess := 1, iDelay := 600,
         xLock := FALSE, xLatch := FALSE, xBuzzer := FALSE);
fbAMInit(iNum := 12, iSeverity := c_AM_ERROR, iProcess := 1, iDelay := 600,
         xLock := FALSE, xLatch := FALSE, xBuzzer := FALSE);

(* 13–18: пускатель напорного не замкнулся — Error, 3 с, ЗАЩЁЛКА (iDelay 60 × 50 мс) *)
fbAMInit(iNum := 13, iSeverity := c_AM_ERROR, iProcess := 1, iDelay := 60,
         xLock := FALSE, xLatch := TRUE, xBuzzer := FALSE);
fbAMInit(iNum := 14, iSeverity := c_AM_ERROR, iProcess := 1, iDelay := 60,
         xLock := FALSE, xLatch := TRUE, xBuzzer := FALSE);
fbAMInit(iNum := 15, iSeverity := c_AM_ERROR, iProcess := 1, iDelay := 60,
         xLock := FALSE, xLatch := TRUE, xBuzzer := FALSE);
fbAMInit(iNum := 16, iSeverity := c_AM_ERROR, iProcess := 1, iDelay := 60,
         xLock := FALSE, xLatch := TRUE, xBuzzer := FALSE);
fbAMInit(iNum := 17, iSeverity := c_AM_ERROR, iProcess := 1, iDelay := 60,
         xLock := FALSE, xLatch := TRUE, xBuzzer := FALSE);
fbAMInit(iNum := 18, iSeverity := c_AM_ERROR, iProcess := 1, iDelay := 60,
         xLock := FALSE, xLatch := TRUE, xBuzzer := FALSE);

(* 19–22: обрыв Pt100 щупы продукта 1–4 — Warning, 3 с (iDelay 60 × 50 мс) *)
fbAMInit(iNum := 19, iSeverity := c_AM_WARNING, iProcess := 1, iDelay := 60,
         xLock := FALSE, xLatch := FALSE, xBuzzer := FALSE);
fbAMInit(iNum := 20, iSeverity := c_AM_WARNING, iProcess := 1, iDelay := 60,
         xLock := FALSE, xLatch := FALSE, xBuzzer := FALSE);
fbAMInit(iNum := 21, iSeverity := c_AM_WARNING, iProcess := 1, iDelay := 60,
         xLock := FALSE, xLatch := FALSE, xBuzzer := FALSE);
fbAMInit(iNum := 22, iSeverity := c_AM_WARNING, iProcess := 1, iDelay := 60,
         xLock := FALSE, xLatch := FALSE, xBuzzer := FALSE);

(* 23: обрыв датчика улицы (0-10 В) — Warning, 3 с (iDelay 60 × 50 мс) *)
fbAMInit(iNum := 23, iSeverity := c_AM_WARNING, iProcess := 1, iDelay := 60,
         xLock := FALSE, xLatch := FALSE, xBuzzer := FALSE);

(* 24–25: обрыв 4-20 мА ПВТ110 (t°, влажность) — Warning, 3 с (iDelay 60 × 50 мс) *)
fbAMInit(iNum := 24, iSeverity := c_AM_WARNING, iProcess := 1, iDelay := 60,
         xLock := FALSE, xLatch := FALSE, xBuzzer := FALSE);
fbAMInit(iNum := 25, iSeverity := c_AM_WARNING, iProcess := 1, iDelay := 60,
         xLock := FALSE, xLatch := FALSE, xBuzzer := FALSE);

(* 26: температура продукта выше макс. — Error, 5 с (iDelay 100 × 50 мс) *)
fbAMInit(iNum := 26, iSeverity := c_AM_ERROR, iProcess := 1, iDelay := 100,
         xLock := FALSE, xLatch := FALSE, xBuzzer := FALSE);

(* 27: влажность ниже минимума — Error, 5 с (iDelay 100 × 50 мс) *)
fbAMInit(iNum := 27, iSeverity := c_AM_ERROR, iProcess := 1, iDelay := 100,
         xLock := FALSE, xLatch := FALSE, xBuzzer := FALSE);

(* 28–33: клапан не закрылся — Warning, 60 с (iDelay g_iValveTime / 20 × 50 мс) *)
fbAMInit(iNum := 28, iSeverity := c_AM_WARNING, iProcess := 1, iDelay := g_iValveTime / 20,
         xLock := FALSE, xLatch := FALSE, xBuzzer := FALSE);
fbAMInit(iNum := 29, iSeverity := c_AM_WARNING, iProcess := 1, iDelay := g_iValveTime / 20,
         xLock := FALSE, xLatch := FALSE, xBuzzer := FALSE);
fbAMInit(iNum := 30, iSeverity := c_AM_WARNING, iProcess := 1, iDelay := g_iValveTime / 20,
         xLock := FALSE, xLatch := FALSE, xBuzzer := FALSE);
fbAMInit(iNum := 31, iSeverity := c_AM_WARNING, iProcess := 1, iDelay := g_iValveTime / 20,
         xLock := FALSE, xLatch := FALSE, xBuzzer := FALSE);
fbAMInit(iNum := 32, iSeverity := c_AM_WARNING, iProcess := 1, iDelay := g_iValveTime / 20,
         xLock := FALSE, xLatch := FALSE, xBuzzer := FALSE);
fbAMInit(iNum := 33, iSeverity := c_AM_WARNING, iProcess := 1, iDelay := g_iValveTime / 20,
         xLock := FALSE, xLatch := FALSE, xBuzzer := FALSE);
END_PROGRAM

PROGRAM ROUTINE
VAR
  fbScaleHost : FB_SCALE_AI;  (* Масштабирование host AI (общий экземпляр для 3 каналов; ValueOut читается через FLT10) *)
  fbScaleRtd : L02_SCALE_AI;  (* Масштабирование L02-RTD (общий экземпляр для 4 щупов; ValueOut читается через FLT10) *)
  fbAMSet : FB_AM_SET;  (* Регистрация условий тревог (34 вызова) *)
  fbAMHas : FB_AM_HAS_ALARMS;  (* Наличие активных тревог *)
  fbAMBlock : FB_AM_IS_BLOCK;  (* Блокирующие тревоги (реле фаз) *)
  fbAMPack : FB_AM_PACK_ALARMS;  (* Упаковка тревог в D550–D552 *)
  fbAMReset : FB_AM_RESET;  (* Сброс тревог (1 с) *)
  xResetCmd : BOOL;  (* Команда сброса (ручной + автосброс) *)
  xResetArmed : BOOL;  (* Автосброс активирован (идёт отсчёт) *)
  iAutoResetCount : INT;  (* Отсчёт до автосброса, с *)
  fbLight : FB_LIGHT;  (* Режимы и световая колонна (единственный ФБ проекта) *)
  PortSettings : DWORD;  (* Параметры порта Modbus (возврат MB_PORT_SETTINGS); задел Modbus slave — по умолчанию отключён *)
  iMbParity : INT;  (* Чётность Modbus из настроек HMI (константа MB_PARITY_*) *)
  iMbStopBit : INT;  (* Стоп-бит Modbus из настроек HMI (константа MB_STOPBIT_*) *)
  iMbBaud : INT;  (* Скорость Modbus из настроек HMI (константа MB_BPS_*) *)
  xMbDummy : BOOL;  (* Фиктивный приёмник результата MB_SLAVE_INIT_PORT2 (требование синтаксиса, см. Modbus.EN.md) *)
END_VAR
(*
  PRG_ROUTINE — программа рутин (Program)
  Проект: автоматизация камеры овощехранилища (ШУК.260726), ПЛК COOLMAY-L02
  Среда: GX Works 2, IEC 61131-3 Structured Text

  Содержит «рутины» — вспомогательные слои, не являющиеся бизнес-логикой:
    1) слой аналоговых входов (код бывшего FB_IO): масштабирование
       7 каналов, коррекции, обрывы; выходы блоков масштабирования (INT, ×10)
       через функцию F_FLT10 → глобальные REAL-переменные AI_f* (для HMI-графиков);
    2) тревоги AlarmManager V212 (код бывшего FB_ALARMS): FB_AM_SET ×34,
       сводные флаги, упаковка для HMI, сброс/автосброс;
    3) световая колонна: вызов ФБ FB_LIGHT (единственный оставшийся ФБ);
    4) Modbus slave (порт 2, RS-485): инициализация для диспетчеризации/PUSH
       (xInit = M8002 или кнопка «Сброс тревог» HMI) — адрес 1, 9600 8N1
       (план §7, задел активирован).

  ФБ FB_IO и FB_ALARMS УДАЛЕНЫ — их код вставлен в эту программу напрямую.
  Бизнес-логика (автомат + приводы) — в программе PRG_MAIN.
  Порядок выполнения программ в задаче: PRG_ROUTINE → PRG_MAIN
  (данные/тревоги до бизнес-логики).

  Тикер TCO_TICKER_50 (TimeControl V2) здесь НЕ вызывается — он настроен
  и работает в отдельной программе TimeControl (план §2).

  Локальные переменные — в PRG_ROUTINE.csv.
 *)

(* Разрешение прерываний (EI) — первая строка каждой программы *)
EI(TRUE);

(* ════════════════════════════════════════════════════════════════
   ЧАСТЬ 1. СЛОЙ АНАЛОГОВЫХ ВХОДОВ (код бывшего FB_IO)
   ════════════════════════════════════════════════════════════════
   - host AI0: температура улицы, датчик 0-10 В (D8030), диапазон
                −50…+50 °C → °C×10, обрыв — по ErrWire (тревога 23);
   - host AI2: температура в камере, ПВТ110 4-20 мА (D8032),
                диапазон −40…+80 °C → °C×10;
   - host AI3: влажность в камере, ПВТ110 4-20 мА (D8033),
                диапазон 5…95 % → %×10;
   - модуль L02-RTD: щупы продукта 1–4 (R23700–R23703) — готовые °C×10;
   - средняя температура продукта по 4 щупам.

   МАСШТАБИРОВАННЫЕ ЗНАЧЕНИЯ: SCALE_AI/L02_SCALE_AI выдают INT в масштабе
   ×10 (например, 245 = 24.5 °C). Для HMI-графиков/трендов TK8100 значения
   переводятся функцией F_FLT10 в REAL (числовое значение сохраняется, ×10;
   деление на 10 — на панели) и пишутся в глобальные REAL-метки AI_f*
   (IO.csv: D0–D15, по 2 слова на REAL).

   СРАВНЕНИЯ В ЛОГИКЕ (тип!):
   - host-каналы (t улицы, t/влажность в камере) — тревоги и автомат читают
     AI_f* (REAL, НАТУРАЛЬНЫЕ единицы: F_FLT10 делит на 10), пороги-настройки
     (g_iToutMin/Max, g_iTpreheat, g_iHmin — INT в масштабе ×10)
     преобразуются функцией F_FLT10: в GX Works 2 IEC ST нет неявного
     преобразования REAL↔INT в операциях сравнения, а INT_TO_REAL без
     деления оставил бы порог в ×10 (неверно);
   - щупы продукта (L02-RTD) — модуль уже выдаёт ГОТОВУЮ температуру °C×10
     в R23700…R23703 (INT), поэтому тревоги 19–22 и 26 сравнивают эти
     регистры напрямую с порогами (INT ↔ INT), без перевода в REAL.

   Коррекция датчиков (настройки HMI, °C×10):
   - g_iCorrTout — датчик улицы;
   - g_iCorrTprod1..4 — щупы продукта 1–4.
   Значение Correction прибавляется к результату (см. Utils V3).
   ВНИМАНИЕ: коррекция щупов применяется в AI_fTProd* (для HMI), но не
   в тревогах 19–22/26 (там — сырые R23700…R23703). Если нужна коррекция
   и в тревогах — сравнивать AI_fTProd* с F_FLT10(порог).

   ОБРЫВЫ host-датчиков определяются по ErrWire SCALE_AI и регистрируются
   (fbAMSet 23–25) СРАЗУ после каждого вызова масштабирования ниже.
   Масштабированные значения пишутся в метки AI_f* (REAL, D0–D15),
   которые читают остальные блоки и HMI.

   Именование: AI_f* — REAL (float), AI_i* — INT(сырые значения).

   Один экземпляр SCALE_AI используется для всех host-каналов,
   один экземпляр L02_SCALE_AI — для всех щупов (см. Utils V3).
 *)


g_xCoolerWorks := DI_CoolerRun;
g_xIsAuto := DI_ModeAuto;
g_xAspirNow := g_iModeDisp = 3;
g_iCurWait := astIntens[g_iIntensity].RECIRC;
g_iCurAsper := astIntens[g_iIntensity].ASPER;
g_xRecycleFlow := (DO_VlvRec1Open OR DO_VlvRec2Open) AND (g_iModeDisp = 2 OR g_iModeDisp = 1);

(* Host AI0: температура улицы, датчик 0-10 В (−50…+50 °C → −500…+500 °C×10).
   Экземпляр fbScaleHost общий для 3 каналов — ErrWire и ValueOut читаем
   СРАЗУ после вызова (следующий вызов их перезапишет).
   Значение SCALE_AI (INT, ×10) через F_FLT10 → глобальная REAL (для HMI). *)
fbScaleHost(iAINum := 0, iSType := STYPE_0_10V, iMin := -500, iMax := 500,
            iCorrection := g_iCorrTout, iFilterTime := 10, iFilterNum := 100);
fbAMSet(iNum := 23, xState := fbScaleHost.xErrWire); (* обрыв 0-10 В *)
AI_fTOutside := F_FLT10(fbScaleHost.iValueOut);

(* Host AI2: температура в камере (ПВТ110, 4-20 мА, −40…+80 °C) *)
fbScaleHost(iAINum := 2, iSType := STYPE_4_20MA, iMin := -400, iMax := 800, iCorrection := g_iTCorrection);
fbAMSet(iNum := 24, xState := fbScaleHost.xErrWire); (* обрыв 4-20 мА, t камеры *)
AI_fTChamber := F_FLT10(fbScaleHost.iValueOut);

(* Host AI3: влажность в камере (ПВТ110, 4-20 мА, 5…95 %) *)
fbScaleHost(iAINum := 3, iSType := STYPE_4_20MA, iMin := 50, iMax := 950);
fbAMSet(iNum := 25, xState := fbScaleHost.xErrWire); (* обрыв 4-20 мА, влажность *)
AI_fHChamber := F_FLT10(fbScaleHost.iValueOut);

(* L02-RTD: щупы температуры продукта 1–4 (готовые °C×10,
   контроль обрыва модулем не выполняется — детекция по значению).
   Экземпляр fbScaleRtd общий для 4 щупов — ValueOut читаем сразу. *)
fbScaleRtd(iAINum := 0, iSType := STYPE_PT100, iCorrection := g_iCorrTprod1);
AI_fTProd1 := F_FLT10(fbScaleRtd.iValueOut);
fbScaleRtd(iAINum := 1, iSType := STYPE_PT100, iCorrection := g_iCorrTprod2);
AI_fTProd2 := F_FLT10(fbScaleRtd.iValueOut);
fbScaleRtd(iAINum := 2, iSType := STYPE_PT100, iCorrection := g_iCorrTprod3);
AI_fTProd3 := F_FLT10(fbScaleRtd.iValueOut);
fbScaleRtd(iAINum := 3, iSType := STYPE_PT100, iCorrection := g_iCorrTprod4);
AI_fTProd4 := F_FLT10(fbScaleRtd.iValueOut);

(* Средняя температура продукта (для HMI, D14; REAL — точнее, чем INT) *)
AI_fTProdAvg := (AI_fTProd1 + AI_fTProd2 + AI_fTProd3 + AI_fTProd4) / 4.0;

(* ════════════════════════════════════════════════════════════════
   ЧАСТЬ 2. ТРЕВОГИ ALARMMANAGER V212 (код бывшего FB_ALARMS)
   ════════════════════════════════════════════════════════════════
   - регистрация условий 34 тревог (FB_AM_SET) — нумерация 0–33, план §5;
   - сводные флаги: g_xAnyAlarm (FB_AM_HAS_ALARMS), g_xAnyBlock (FB_AM_IS_BLOCK);
   - упаковка тревог для HMI: D550 (биты 0–15), D551 (биты 16–31), D552 (биты 32–33);
   - сброс: ручной (кнопка HMI g_xAlarmResetHmi) и автосброс
     (g_xAutoReset = TRUE, через g_iAutoResetDelay минут).

   Полярности входов (проверить при пусконаладке, см. вопросы §1.3):
   - концевики клапанов «закрыт» — контакт НО: «закрыт» = вход 1,
     «не закрыт» = вход 0 (тревоги 28–33);
   - концевики клапанов «открыт» — плк.txt указывает НО («открыт» = вход 1,
     «не открыт» = вход 0), но тревоги 1–6 ниже всё ещё закодированы под
     прежнюю НЗ-полярность — привести к НО после подтверждения на стенде;
   - РД-ДД200 — контакт НЗ: «поток есть» = вход 0, «нет потока» = вход 1.

   Обрывы host-датчиков (23–25) регистрируются по fbScaleHost.xErrWire
   СРАЗУ после масштабирования в части 1 и здесь НЕ повторяются.
   Обрыв щупов Pt100 (19–22) — по значению ≤ −1900 (модуль L02-RTD
   контроля обрыва не имеет, см. план §4, п.5).
 *)

(* ── Регистрация условий тревог ───────────────────────────────── *)
(* 0: реле контроля фаз — ошибка фазировки *)
fbAMSet(iNum := 0, xState := NOT DI_PhaseFault);

(* 1–6:клапан не открылся — командв «открыть» подана,
   а концевик «открыт» (НО) не сработал. НО: DI_*Open = 1 — клапан открыт,
   0 — закрыт.*)
fbAMSet(iNum := 1, xState := DO_VlvIn1Open AND NOT DI_VlvIn1Open);
fbAMSet(iNum := 2, xState := DO_VlvIn2Open AND NOT DI_VlvIn2Open);
fbAMSet(iNum := 3, xState := DO_VlvOut1Open AND NOT DI_VlvOut1Open);
fbAMSet(iNum := 4, xState := DO_VlvOut2Open AND NOT DI_VlvOut2Open);
fbAMSet(iNum := 5, xState := DO_VlvRec1Open AND NOT DI_VlvRec1Open);
fbAMSet(iNum := 6, xState := DO_VlvRec2Open AND NOT DI_VlvRec2Open);

(* 28–33: клапан не закрылся — команды «открыть» нет (пружина закрывает),
   а концевик «закрыт» (НО) не сработал. НО: DI_*Close = 1 — клапан закрыт,
   0 — не закрыт.*)
fbAMSet(iNum := 28, xState := NOT DO_VlvIn1Open AND NOT DI_VlvIn1Close);
fbAMSet(iNum := 29, xState := NOT DO_VlvIn2Open AND NOT DI_VlvIn2Close);
fbAMSet(iNum := 30, xState := NOT DO_VlvOut1Open AND NOT DI_VlvOut1Close);
fbAMSet(iNum := 31, xState := NOT DO_VlvOut2Open AND NOT DI_VlvOut2Close);
fbAMSet(iNum := 32, xState := NOT DO_VlvRec1Open AND NOT DI_VlvRec1Close);
fbAMSet(iNum := 33, xState := NOT DO_VlvRec2Open AND NOT DI_VlvRec2Close);


(* 7–12: нет потока воздуха, напорные вентиляторы 1–6 *)
fbAMSet(iNum := 7, xState := DO_FanH1 AND NOT DI_Flow1);
fbAMSet(iNum := 8, xState := DO_FanH2 AND NOT DI_Flow2);
fbAMSet(iNum := 9, xState := DO_FanH3 AND NOT DI_Flow3);
fbAMSet(iNum := 10, xState := DO_FanH4 AND NOT DI_Flow4);
fbAMSet(iNum := 11, xState := DO_FanH5 AND NOT DI_Flow5);
fbAMSet(iNum := 12, xState := DO_FanH6 AND NOT DI_Flow6);

(* 13–18: пускатель напорного вентилятора не замкнулся (ОС не пришла) *)
fbAMSet(iNum := 13, xState := DO_FanH1 AND NOT DI_FanHFb1);
fbAMSet(iNum := 14, xState := DO_FanH2 AND NOT DI_FanHFb2);
fbAMSet(iNum := 15, xState := DO_FanH3 AND NOT DI_FanHFb3);
fbAMSet(iNum := 16, xState := DO_FanH4 AND NOT DI_FanHFb4);
fbAMSet(iNum := 17, xState := DO_FanH5 AND NOT DI_FanHFb5);
fbAMSet(iNum := 18, xState := DO_FanH6 AND NOT DI_FanHFb6);

(* 19–22: обрыв Pt100 — щупы продукта 1–4 (значение ≤ −190 °C).
   Модуль L02-RTD выдаёт ГОТОВУЮ температуру в R23700…R23703 (INT, °C×10) —
   сравниваем её напрямую (без перевода в REAL), тип INT совпадает. *)
fbAMSet(iNum := 19, xState := R23700 <= -1900);
fbAMSet(iNum := 20, xState := R23701 <= -1900);
fbAMSet(iNum := 21, xState := R23702 <= -1900);
fbAMSet(iNum := 22, xState := R23703 <= -1900);

(* 26: температура продукта выше максимума (любой из 4 щупов) —
   сравнение по готовым значениям модуля R23700…R23703 (INT, °C×10) *)
fbAMSet(iNum := 26, xState := (R23700 > g_iTprodMax) OR
                              (R23701 > g_iTprodMax) OR
                              (R23702 > g_iTprodMax) OR
                              (R23703 > g_iTprodMax));

(* 27: влажность ниже минимума (исключая обрыв 4-20 мА).
   AI_fHChamber — REAL в натуральных единицах (F_FLT10 делит на 10),
   g_iHmin — INT в масштабе ×10 → порог переводится функцией F_FLT10
   (в GX Works 2 нет неявного REAL↔INT в сравнениях). *)
fbAMSet(iNum := 27, xState := AI_fHChamber < F_FLT10(g_iHmin));

(* ── Сводные флаги для логики и HMI ──────────────────────────── *)
fbAMHas(iProcessNum := 0, iSeverity := 0, Q := g_xAnyAlarm, AC := g_iAlarmCount);
fbAMBlock(iProcessNum := 0, iSeverity := 0, Q := g_xAnyBlock);

(* ── Упаковка тревог для HMI: M600 - 0, M601 - 1, ... ── *)
fbAMPack(DNUM := 600, PD := c_AM_PACK_M);

(* ── Сброс тревог ────────────────────────────────────────────── *)
(* FB_AM_RESET удерживает сигнал сброса 1 с (см. AlarmManager V212) *)
fbAMReset(IN := g_xAlarmResetHmi, AutoReset := g_iAutoResetDelay * 60);

(* ════════════════════════════════════════════════════════════════
   ЧАСТЬ 3. СВЕТОВАЯ КОЛОННА (ФБ FB_LIGHT)
   ════════════════════════════════════════════════════════════════
   Выбор режима и индикация по плану §6.7. FB_LIGHT — единственный
   оставшийся в проекте функциональный блок (кроме библиотечных).
 *)
fbLight();

(* Состояние вентияторов
0=выкл, 1=вкл, 2=тревога *)
g_iFun1State := 0;
MOV(DO_FanH1, 1, g_iFun1State);
MOV(AM_ALARMS[13].Alarm, 2, g_iFun1State);

g_iFun2State := 0;
MOV(DO_FanH2, 1, g_iFun2State);
MOV(AM_ALARMS[14].Alarm, 2, g_iFun2State);

g_iFun3State := 0;
MOV(DO_FanH3, 1, g_iFun3State);
MOV(AM_ALARMS[15].Alarm, 2, g_iFun3State);

g_iFun4State := 0;
MOV(DO_FanH4, 1, g_iFun4State);
MOV(AM_ALARMS[16].Alarm, 2, g_iFun4State);

g_iFun5State := 0;
MOV(DO_FanH5, 1, g_iFun5State);
MOV(AM_ALARMS[17].Alarm, 2, g_iFun5State);

g_iFun6State := 0;
MOV(DO_FanH6, 1, g_iFun6State);
MOV(AM_ALARMS[18].Alarm, 2, g_iFun6State);

g_iFun7State := 0;
MOV(DO_FanR1, 1, g_iFun7State);

g_iFun8State := 0;
MOV(DO_FanR2, 1, g_iFun8State);

g_iFun9State := 0;
MOV(DO_FanR3, 1, g_iFun9State);

g_iFun10State := 0;
MOV(DO_FanR4, 1, g_iFun10State);

(* ════════════════════════════════════════════════════════════════
   ЧАСТЬ 4. MODBUS SLAVE — ПОРТ 2 (RS-485) ════════════════════════
   Инициализация слейва для диспетчеризации / PUSH-интеграции:
   внешний мастер (шлюз/облако) опрашивает ПЛК по Modbus RTU.
   - порт 2 (клеммник RS-485), адрес slave = 1, 9600 8N1;
   - xInit (вход функции MB_SLAVE_INIT_PORT2): M8002 (первый скан ПЛК)
     ИЛИ кнопка HMI «Сброс тревог» (g_xAlarmResetHmi). По Modbus.EN.md
     слейв (пере)инициализируется по КАЖДОМУ фронту xInit, поэтому
     оборачивать вызов в IF M8002 НЕ нужно — условие передаётся во вход;
   - адресация регистров слейва — по умолчанию библиотеки (прямой доступ
     к D-регистрам ПЛК); буфер D600–D800 (план §7) нужен только для режима
     Master (MB_PROCESS_50), если он понадобится позже;
   - PortSettings — параметры порта (DWORD, возврат MB_PORT_SETTINGS);
   - xMbDummy — фиктивный приёмник результата функции: по Modbus.EN.md
     вызов функции-выражения как оператора требует присваивания слева.

   ⚠ Полярность: для включения Modbus slave порт 2 ПЛК должен быть
   настроен на RS-485 (аппаратно), адрес/скорость — выше.
 *)
PortSettings := MB_PORT_SETTINGS(MB_PARITY_NONE, MB_STOPBIT_1, MB_BPS_9600);
xMbDummy := MB_SLAVE_INIT_PORT2(M8002 OR g_xMbApply, g_iMbAddr, PortSettings);
END_PROGRAM

FUNCTION_BLOCK FB_LIGHT
VAR
  xAspMode : BOOL;  (* Идёт аспирация (g_iModeDisp = 2) *)
  xRed : BOOL;  (* Сигнал красной лампы *)
  xGreen : BOOL;  (* Сигнал зелёной лампы *)
END_VAR
(*
  MODE — выбор режима и световая колонна (FB)
  Режим по переключателю (приоритет — «Продувка», план §6.1):
    X00=0, X01=0 → Выключено (0)
    X00=1        → Авто (1)
    X01=1        → Продувка (3) — приоритет, даже если X00=1

  Грубый режим записывается в g_iModeCoarse (D222); детальный
  (Рециркуляция/Аспирация) формирует PROCESS в g_iModeDisp (D200).

  Световая колонна по плану §6.7 (мигание — M8013, 0.5 с / 0.5 с):
    Выключено        🔴 off        🟢 off
    Продувка         🔴 on         🟢 on
    Авто-рециркуляция 🔴 миг.(трев.) 🟢 on
    Авто-аспирация   🔴 миг.(трев.) 🟢 миг.
    Тревоги (любой режим) 🔴 мигает

  Экземпляр ФБ: fbMode (MAIN.csv). Локальные переменные — в mode.csv.
*)

(* Идёт ли аспирация (детальный режим из PROCESS, прошлый скан) *)
xAspMode := (g_iModeDisp = 2);

(* Красный: мигает при любой активной тревоге, горит в Продувке *)
IF g_xAnyAlarm THEN
    xRed := M8013;
ELSIF g_iModeCoarse = 3 THEN
    xRed := TRUE;
ELSE
    xRed := FALSE;
END_IF;

(* Зелёный *)
IF g_iModeCoarse = 3 THEN
    xGreen := TRUE;                  (* Продувка — горит постоянно *)
ELSIF g_iModeCoarse = 1 OR g_xManualAspActive THEN
    IF xAspMode THEN
        xGreen := M8013;             (* Аспирация — мигает *)
    ELSE
        xGreen := TRUE;              (* Рециркуляция — горит *)
    END_IF;
ELSE
    xGreen := FALSE;                 (* Выключено — выключена *)
END_IF;

(* Выходы световой колонны *)
DO_LampRed := xRed;
DO_LampGreen := xGreen;
END_FUNCTION_BLOCK
